Yaskawa INFORM job: TCP_SHORT_SPIKE(FRONIUS).JBI

/JOB
//NAME TCP_SHORT_SPIKE(FRONIUS)
///FOLDERNAME INNE
//POS
///NPOS 15,15,0,0,0,0
///TOOL 0
///POSTYPE PULSE
///PULSE
C00000=-4583,5642,89476,4172,104763,40737
C00001=51552,-20253,55040,3434,103292,51107
C00002=123138,-21385,54332,3464,103143,51107
C00003=159941,-23787,51536,4061,104329,41262
C00004=218457,-23942,51455,4750,104259,41509
C00005=-234857,-7102,73443,5072,104923,43998
C00006=-153018,-2614,78799,5247,103831,50699
C00007=-123869,-4125,76427,5422,105682,39334
C00008=-40112,-13409,63505,-3433,107469,-25610
C00009=-58981,-52163,17422,-3697,97286,-35739
C00010=-170551,-40692,30621,-3142,100533,-41102
C00011=-222678,-73071,-848,-828,90512,-10144
C00012=-33739,-101128,-19534,4446,67644,31852
C00013=35637,-71876,-568,2810,84711,58622
C00014=-5687,-47768,22058,4093,98617,38654
BC00000=234605,127399,695028
BC00001=234605,127399,695029
BC00002=234605,127399,695029
BC00003=234605,127399,695029
BC00004=234605,127399,695029
BC00005=234604,127399,695026
BC00006=234605,127399,695029
BC00007=234605,127399,695029
BC00008=234605,127399,695029
BC00009=234605,127399,695029
BC00010=234605,127399,695029
BC00011=234605,127399,695029
BC00012=234605,127399,695029
BC00013=234605,127399,695027
BC00014=234605,127399,695029
//INST
///DATE 2023/10/04 15:16
///ATTR SC,RW
///GROUP1 RB1,BS1
NOP
MOVJ C00000 BC00000 VJ=0.78
MOVJ C00001 BC00001 VJ=0.78
MOVJ C00002 BC00002 VJ=0.78
MOVJ C00003 BC00003 VJ=0.78
MOVJ C00004 BC00004 VJ=0.78
MOVJ C00005 BC00005 VJ=0.78
MOVJ C00006 BC00006 VJ=0.78
MOVJ C00007 BC00007 VJ=0.78
MOVJ C00008 BC00008 VJ=0.78
MOVJ C00009 BC00009 VJ=0.78
MOVJ C00010 BC00010 VJ=0.78
MOVJ C00011 BC00011 VJ=0.78
MOVJ C00012 BC00012 VJ=0.78
MOVJ C00013 BC00013 VJ=0.78
MOVJ C00014 BC00014 VJ=0.78
END
